# EPICS substitutions: tpmacApp/Db/autohome.substitutions
file "$(EPICS_BASE)/db/autohome.db"
{

pattern
{SYS,              DEV,                 PLC,  PORT  }
{"XF:23ID2-OP",  "{Slt:1-Ax:T}",      8,     P0    }
{"XF:23ID2-OP",  "{Slt:1-Ax:B}",      9,     P0    }
{"XF:23ID2-OP",  "{Slt:1-Ax:O}",      10,    P0    }
{"XF:23ID2-OP",  "{Slt:1-Ax:I}",      11,    P0    }
{"XF:23ID2-BI",  "{Diag:Slt1-Ax:Y}",  15,    P0    }
}
